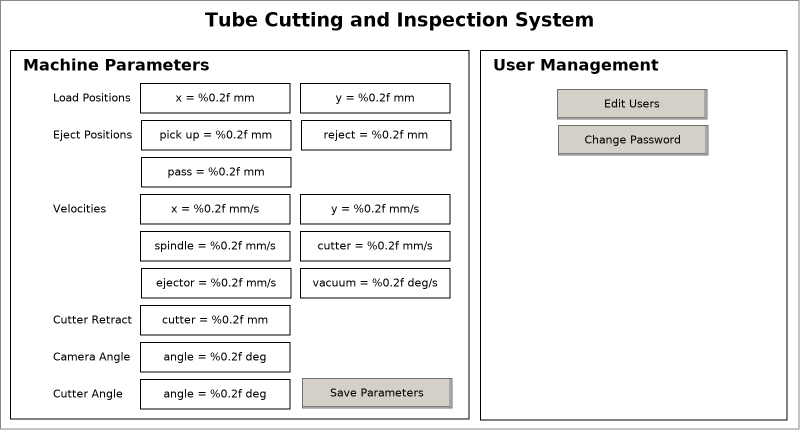
VISUALIZATION MachineSettings  // 800x430
    Label (0,5 800x30), "Tube Cutting and Inspection System"
    Rectangle (10,50 459x369)
    Button (302,378 150x30), "Save Parameters"
        OnMouseClick: execute { MAIN.bSave := TRUE; }
    Label (50,83 90x30), "Load Positions"
    Rectangle (140,83 150x30), "x = %0.2f mm", text variable: MAIN.fbSlitter.Mandrel._hmiParameters.loadPositionX
        OnMouseClick: write MAIN.fbSlitter.Mandrel._hmiParameters.loadPositionX via Default, title 'Load Position X'
    Rectangle (300,83 150x30), "y = %0.2f mm", text variable: MAIN.fbSlitter.Mandrel._hmiParameters.loadPositionY
        OnMouseClick: write MAIN.fbSlitter.Mandrel._hmiParameters.loadPositionY via Default, title 'Load Position Y'
    Label (50,194 90x30), "Velocities"
    Rectangle (140,194 150x30), "x = %0.2f mm/s", text variable: MAIN.fbSlitter.Mandrel._hmiParameters.velocityX
        OnMouseClick: write MAIN.fbSlitter.Mandrel._hmiParameters.VelocityX via Default, title 'X Axis Velocity'
    Rectangle (300,194 150x30), "y = %0.2f mm/s", text variable: MAIN.fbSlitter.Mandrel._hmiParameters.velocityY
        OnMouseClick: write MAIN.fbSlitter.Mandrel._hmiParameters.velocityY via Default, title 'Y Axis Velocity'
    Rectangle (140,231 150x30), "spindle = %0.2f mm/s", text variable: MAIN.fbSlitter.Mandrel._hmiParameters.spindleVelocity
        OnMouseClick: write MAIN.fbSlitter.Mandrel._hmiParameters.spindleVelocity via Default, title 'Spindle Velocity'
    Rectangle (300,231 150x30), "cutter = %0.2f mm/s", text variable: MAIN.fbSlitter.Cutter._hmiParameters.cutVelocity
        OnMouseClick: write MAIN.fbSlitter.Cutter._hmiParameters.cutVelocity via Default, title 'Cutter Axis Velocity'
    Label (50,305 90x30), "Cutter Retract"
    Rectangle (140,305 150x30), "cutter = %0.2f mm", text variable: MAIN.fbSlitter.Cutter._hmiParameters.retractPosition
        OnMouseClick: write MAIN.fbSlitter.Cutter._hmiParameters.retractPosition via Default, title 'Cutter Retract Position'
    Rectangle (140,342 150x30), "angle = %0.2f deg", text variable: MAIN.fbSlitter.Camera._hmiParameters.angle
        OnMouseClick: write MAIN.fbSlitter.Camera._hmiParameters.angle via Default, title 'Camera Angle'
    Label (50,342 90x30), "Camera Angle"
    Label (20,50 189x30), "Machine Parameters"
    Rectangle (140,379 150x30), "angle = %0.2f deg", text variable: MAIN.fbSlitter.Mandrel._hmiParameters.spindleOffset
        OnMouseClick: write MAIN.fbSlitter.Mandrel._hmiParameters.spindleOffset via Default, title 'Cutter to Camera Angular Offset'
    Label (50,379 90x30), "Cutter Angle"
    Rectangle (480,50 307x370)
    Label (490,50 189x30), "User Management"
    Button (557,89 150x30), "Edit Users"
        OnMouseClick: VisuUserMgmt Type=OpenUserConfiguration
    Button (558,125 150x30), "Change Password"
        OnMouseClick: VisuUserMgmt Type=ChangeUserPassword
    Rectangle (141,268 150x30), "ejector = %0.2f mm/s", text variable: MAIN.fbSlitter.Ejector._hmiParameters.ejectVelocity
        OnMouseClick: write MAIN.fbSlitter.Ejector._hmiParameters.ejectVelocity via Default, title 'Ejector Axis Velocity'
    Label (50,120 90x30), "Eject Positions"
    Rectangle (141,120 150x30), "pick up = %0.2f mm", text variable: MAIN.fbSlitter.Ejector._hmiParameters.ejectPositionHome
        OnMouseClick: write MAIN.fbSlitter.Ejector._hmiParameters.ejectPositionHome via Default, title 'Eject Pick Up Position'
    Rectangle (301,120 150x30), "reject = %0.2f mm", text variable: MAIN.fbSlitter.Ejector._hmiParameters.ejectPositionFail
        OnMouseClick: write MAIN.fbSlitter.Ejector._hmiParameters.ejectPositionFail via Default, title 'Reject Position'
    Rectangle (141,157 150x30), "pass = %0.2f mm", text variable: MAIN.fbSlitter.Ejector._hmiParameters.ejectPositionPass
        OnMouseClick: write MAIN.fbSlitter.Ejector._hmiParameters.ejectPositionPass via Default, title 'Eject Pass Position'
    Rectangle (300,268 150x30), "vacuum = %0.2f deg/s", text variable: MAIN.fbSlitter.Mandrel._hmiParameters.vacuumVelocity
        OnMouseClick: write MAIN.fbSlitter.Mandrel._hmiParameters.vacuumVelocity via Default, min 0, max 360, title 'Vacuum Axis Velocity'
END_VISUALIZATION

(* stored: Version 1.1.0.1, ProductVersion 3.1.4024.9
   Visu MachineSettings: Id {510e3b73-14a6-4864-8bbe-3d182f383fda} *)
